DATA_BLOCK "滑台伺服S200"   // DB8, Motion_DB
// stored: InstanceOfName TO_PositioningAxis, OfSystemLibElement TO_PositioningAxis, OfSystemLibVersion 6.0
TO_PositioningAxis   // technology object, version 6.0
// stored: Connection Interface Actor, InputAddress 1032, OutputAddress 1056
// stored: Connection Interface Sensor[1], InputAddress 1032, OutputAddress 1056, SensorIndexInActorTelegram 1
   // // inherited from TO_SpeedAxis
   // // inherited from TO_Axis
   // // inherited from TO_Object
   // VAR
   //    Actor : TO_Struct_Actor;
   // END_VAR
   // VAR
   //    Position { ExternalWritable := 'False'} : LReal;
   //    ActualPosition { ExternalWritable := 'False'} : LReal;
   //    ActualVelocity { ExternalWritable := 'False'} : LReal;
   //    ActualAcceleration { ExternalWritable := 'False'} : LReal;
   //    OperativeSensor { ExternalWritable := 'False'} : UDInt;
   //    ModuloCycle { ExternalWritable := 'False'} : DInt;
   //    ActualModuloCycle { ExternalWritable := 'False'} : DInt;
   //    Clamping { S7_SetPoint := 'True'} : TO_Struct_Clamping;
   //    Sensor { S7_SetPoint := 'True'} : Array[1..4] of TO_Struct_Sensor;
   //    Extrapolation { S7_SetPoint := 'True'} : TO_Struct_Extrapolation;
   //    Mechanics { S7_SetPoint := 'True'} : TO_Struct_Mechanics;
   //    Properties { ExternalWritable := 'False'; S7_SetPoint := 'True'} : TO_Struct_Properties;
   //    Modulo { S7_SetPoint := 'True'} : TO_Struct_Modulo;
   //    PositionLimits_SW { S7_SetPoint := 'True'} : TO_Struct_PositionLimitsSW;
   //    PositionLimits_HW { S7_SetPoint := 'True'} : TO_Struct_PositionLimitsHW;
   //    Homing { S7_SetPoint := 'True'} : TO_Struct_Homing;
   //    PositionControl { S7_SetPoint := 'True'} : TO_Struct_PositionControl;
   //    DynamicAxisModel { S7_SetPoint := 'True'} : TO_Struct_DynamicAxisModel;
   //    FollowingError { S7_SetPoint := 'True'} : TO_Struct_FollowingError;
   //    CrossPlcSynchronousOperation { S7_SetPoint := 'True'} : TO_Struct_CrossPlcSynchronousOperation;
   //    PositioningMonitoring { S7_SetPoint := 'True'} : TO_Struct_PositioningMonitoring;
   //    StandstillSignal { S7_SetPoint := 'True'} : TO_Struct_StandstillSignal;
   //    StatusPositioning { ExternalWritable := 'False'; S7_SetPoint := 'True'} : TO_Struct_StatusPositioning;
   //    StatusServo { ExternalWritable := 'False'; S7_SetPoint := 'True'} : TO_Struct_StatusServo;
   //    StatusProvidedLeadingValue { ExternalWritable := 'False'; S7_SetPoint := 'True'} : TO_Struct_StatusProvidedLeadingValue;
   //    StatusSensor { ExternalWritable := 'False'; S7_SetPoint := 'True'} : Array[1..4] of TO_Struct_StatusSensor;
   //    StatusExtrapolation { ExternalWritable := 'False'; S7_SetPoint := 'True'} : TO_Struct_StatusExtrapolation;
   //    StatusKinematicsMotion { ExternalWritable := 'False'; S7_SetPoint := 'True'} : TO_Struct_StatusKinematicsMotion;
   // END_VAR
BEGIN
   Actor.DataAdaption := 1;
   Actor.Interface.AddressIn.RID := 16#208072a;
   Actor.Interface.AddressIn.AREA := 16#81;
   Actor.Interface.AddressIn.OFFSET := 2080;
   Actor.Interface.AddressOut.RID := 16#208072b;
   Actor.Interface.AddressOut.AREA := 16#82;
   Actor.Interface.AddressOut.OFFSET := 2080;
   Actor.Interface.EnableTorqueData := true;
   Actor.Interface.TorqueDataAddressIn.RID := 16#2080742;
   Actor.Interface.TorqueDataAddressIn.AREA := 16#81;
   Actor.Interface.TorqueDataAddressIn.OFFSET := 2240;
   Actor.Interface.TorqueDataAddressOut.RID := 16#2080743;
   Actor.Interface.TorqueDataAddressOut.AREA := 16#82;
   Actor.Interface.TorqueDataAddressOut.OFFSET := 2240;
   Actor.DriveParameter.ReferenceSpeed := 6500.0;
   Actor.DriveParameter.MaxSpeed := 6500.0;
   Actor.DriveParameter.ReferenceTorque := 1.24195;
   Sensor[1]."Type" := 2;
   Sensor[1].DataAdaption := 1;
   Sensor[1].Interface.AddressIn.RID := 16#208072a;
   Sensor[1].Interface.AddressIn.AREA := 16#81;
   Sensor[1].Interface.AddressIn.OFFSET := 2080;
   Sensor[1].Interface.AddressOut.RID := 16#208072b;
   Sensor[1].Interface.AddressOut.AREA := 16#82;
   Sensor[1].Interface.AddressOut.OFFSET := 2080;
   Sensor[1].Parameter.StepsPerRevolution := 1024;
   Sensor[1].Parameter.FineResolutionXist1 := 0;
   Sensor[1].Parameter.FineResolutionXist2 := 0;
   Sensor[1].ActiveHoming.Mode := 2;
   Sensor[1].ActiveHoming.DigitalInputAddress.RID := 16#2000001;
   Sensor[1].ActiveHoming.DigitalInputAddress.AREA := 16#81;
   Sensor[1].ActiveHoming.DigitalInputAddress.OFFSET := 3;
   PositionLimits_HW.Active := true;
   PositionLimits_HW.MinSwitchAddress.RID := 16#2000001;
   PositionLimits_HW.MinSwitchAddress.AREA := 16#81;
   PositionLimits_HW.MinSwitchAddress.OFFSET := 4;
   PositionLimits_HW.MaxSwitchAddress.RID := 16#2000001;
   PositionLimits_HW.MaxSwitchAddress.AREA := 16#81;
   PositionLimits_HW.MaxSwitchAddress.OFFSET := 5;
   PositionControl.EnableDSC := true;
   Actor.Interface.EnableTorqueData := True;
   _Sensor[1].ActiveHoming.DigitalInputAddress := S200原点信号;
   _PositionLimits_HW.MinSwitchAddress := S200正限位;
   _PositionLimits_HW.MaxSwitchAddress := S200负限位;
   _Actor.Interface.Telegram := 105;
   _Actor.DataAdaptionOffline := True;
   _Sensor[1].Interface.Telegram := 105;
   _Sensor[1].DataAdaptionOffline := True;
END_DATA_BLOCK
